(* CoDeSys 2.3.9.41 project: pns.pro *)
(* Libraries: STANDARD.LIB 4.10.05 10:14:46, IECSFC.LIB 13.4.06 14:51:28, SYSLIBTIME.LIB 20.2.06 13:31:16, SYSTASKINFO.LIB 20.2.06 13:31:38, ANALYZATION.LIB 5.10.99 08:05:06, SYSLIBCALLBACK.LIB 20.2.06 13:31:08, PID_Regulators.lib 28.12.06 17:47:54 *)

(* PLC configuration (modules and I/O channels)
Discrete input 6 bit [ID100] node 0, in %IB0 out %QB0 {Filtrationtime = 10; Filtrationtime = 10; Filtrationtime = 10; Filtrationtime = 10; Filtrationtime = 10; Filtrationtime = 10; Visibility = No; PinCount = 6; WatchDogPeriod = 1000; PollPeriod = 1}
  DI_ekmLower AT %IX0.0 [BitInput]
  DI_ekmUpper AT %IX0.1 [BitInput]
  DI_pmp1_auto AT %IX0.2 [BitInput]
  DI_pmp2_auto AT %IX0.3 [BitInput]
  DI_pmp3_auto AT %IX0.4 [BitInput]
  DI_fcAlarm AT %IX0.5 [BitInput]
Discrete output 4 bit [ID101] node 1, in %IB1 out %QB1 {PinCount = 4; SafeValueBool = FALSE; SafeValueBool = FALSE; SafeValueBool = FALSE; SafeValueBool = FALSE; Visibility = No}
  DO_fc_on AT %QX1.0 [BitOutput]
  DO_fc_run AT %QX1.1 [BitOutput]
  DO_lamp_fcAlarm AT %QX1.2 [BitOutput]
  DO_lamp_dryHod AT %QX1.3 [BitOutput]
Special output [ID104] node 2, in %IB2 out %QB2 {Visibility = No; PinCount = 1}
  AT %QX2.0 [BitOutput] Special output
Unifed signal sensor [ID700] node 3, in %IB3 out %QB3 {Type_of_sensor700 = IT_0_20; measure_interval = 0.5; ainlow = 0; ainhigh = 20; first_cor_point = 0; first_delta = 0; second_cor_point = 0; second_delta = 0; third_cor_point = 0; third_delta = 0; Visibility = No}
  AI_pres AT %ID3.0 [FloatInput] Value
  cirTime AT %IW3.1 [WordInput] Circular time
  Analog Input [ID107] node 0, in %IB3.0 out %QB3.0
Unifed signal sensor [ID700] node 4, in %IB4 out %QB4 {Type_of_sensor700 = IT_0_20; measure_interval = 0.5; ainlow = 0; ainhigh = 20; first_cor_point = 0; first_delta = 0; second_cor_point = 0; second_delta = 0; third_cor_point = 0; third_delta = 0; Visibility = No}
  AT %ID4.0 [FloatInput] Value
  AT %IW4.1 [WordInput] Circular time
  Analog Input [ID107] node 0, in %IB4.0 out %QB4.0
Unifed signal sensor [ID700] node 5, in %IB5 out %QB5 {Type_of_sensor700 = IT_0_20; measure_interval = 0.5; ainlow = 0; ainhigh = 20; first_cor_point = 0; first_delta = 0; second_cor_point = 0; second_delta = 0; third_cor_point = 0; third_delta = 0; Visibility = No}
  AT %ID5.0 [FloatInput] Value
  AT %IW5.1 [WordInput] Circular time
  Analog Input [ID107] node 0, in %IB5.0 out %QB5.0
Unifed signal sensor [ID700] node 6, in %IB6 out %QB6 {Type_of_sensor700 = IT_0_20; measure_interval = 0.5; ainlow = 0; ainhigh = 20; first_cor_point = 0; first_delta = 0; second_cor_point = 0; second_delta = 0; third_cor_point = 0; third_delta = 0; Visibility = No}
  AT %ID6.0 [FloatInput] Value
  AT %IW6.1 [WordInput] Circular time
  Analog Input [ID107] node 0, in %IB6.0 out %QB6.0
Analog output [ID106] node 7, in %IB7 out %QB7 {DAC_Type = Voltage 0-10 B; Analog_offset_correction = 0; Analog_full_range_correction = 0; SafeValueFloat = 0; Visibility = No}
  AO_ref AT %QD7.0 [FloatOutput] Value
Analog output [ID106] node 8, in %IB8 out %QB8 {DAC_Type = Voltage 0-10 B; Analog_offset_correction = 0; Analog_full_range_correction = 0; SafeValueFloat = 0; Visibility = No}
  AT %QD8.0 [FloatOutput] Value
ModBus (Master) [MODBUS_MASTER_ID450] node 9, in %IB9 out %QB9 {Visibility = No}
  AT %QD9.0 [DWordOutput] Last address
  AT %QW9.1 [WordOutput] Last error
  RS-485-1 [COM1_USART] node 0, in %IB9.0 out %QB9.0 {CommunicationSpeed = 19200; Parity = NO PARITY CHECK; BitLength = 8 bits; StopLength = One stop bit; InterfaceType = RS485; FrameOriented = RTU; Timeout = 0; Visibility = No}
  Universal Modbus device [ID2000] node 1, in %IB9.1 out %QB9.1 {ModuleIP = 10:0:0:223; ServiceTimeout = 150; TCPport = 502; NetMode = Serial; ModuleSlaveAddress = 2; RequestType = By poll time; PeriodOfService = 500; Visibility = No; RepeatCounter = 0; ByteSequence = Trace_mode}
    AT %QB9.1.0 [ComChannel] Command (0xff - Start)
PLC100_DI AT %IW9.1.0.0 [WordInput]
PLC100_DO AT %QW9.1.1.0 [WordOutput]
TCP [TCP_ID221] node 0, in %IB10.0.0 out %QB10.0.0 {RemotePort = 502; Visibility = No}
ktp_INPUT AT %QW10.1.0 [WordOutput] setTime, kaReset
ktp_OUTPUT AT %QW10.2.0 [WordOutput] pmp1,pmp2,pmp3,EKM,alarm,auto1,auto2,auto3
ktp_pressure AT %QW10.3.0 [WordOutput]
ktp_presStartDelta AT %QW10.4.0 [WordOutput]
ktp_presStopDelta AT %QW10.5.0 [WordOutput]
ktp_daySetpoint AT %QW10.6.0 [WordOutput]
ktp_nightSetpoint AT %QW10.7.0 [WordOutput]
ktp_finishSetpoint AT %QW10.8.0 [WordOutput]
ktp_pres4ma AT %QW10.9.0 [WordOutput]
ktp_pres20ma AT %QW10.10.0 [WordOutput]
ktp_startReserveDelay AT %QW10.11.0 [WordOutput]
ktp_stopReserveDelay AT %QW10.12.0 [WordOutput]
ktp_barToStartDirect AT %QW10.13.0 [WordOutput]
ktp_mainPmp AT %QW10.14.0 [WordOutput]
ktp_prop AT %QW10.15.0 [WordOutput]
ktp_integ AT %QW10.16.0 [WordOutput]
ktp_diff AT %QW10.17.0 [WordOutput]
ktp_integMin AT %QW10.18.0 [WordOutput]
ktp_integMax AT %QW10.19.0 [WordOutput]
ktp_dryHodDelay AT %QW10.20.0 [WordOutput]
ktp_aType_1 AT %QW10.21.0 [WordOutput]
ktp_aType_2 AT %QW10.22.0 [WordOutput]
ktp_aType_3 AT %QW10.23.0 [WordOutput]
ktp_aTime_1 AT %QW10.24.0 [WordOutput]
ktp_aTime_2 AT %QW10.25.0 [WordOutput]
ktp_aTime_3 AT %QW10.26.0 [WordOutput]
ktp_aDate_1 AT %QW10.27.0 [WordOutput]
ktp_aDate_2 AT %QW10.28.0 [WordOutput]
ktp_aDate_3 AT %QW10.29.0 [WordOutput]
ktp_aPres_1 AT %QW10.30.0 [WordOutput]
ktp_aPres_2 AT %QW10.31.0 [WordOutput]
ktp_aPres_3 AT %QW10.32.0 [WordOutput]
ktp_aSetpoint_1 AT %QW10.33.0 [WordOutput]
ktp_aSetpoint_2 AT %QW10.34.0 [WordOutput]
ktp_aSetpoint_3 AT %QW10.35.0 [WordOutput]
ktp_aFreq_1 AT %QW10.36.0 [WordOutput]
ktp_aFreq_2 AT %QW10.37.0 [WordOutput]
ktp_aFreq_3 AT %QW10.38.0 [WordOutput]
ktp_aCurr_1 AT %QW10.39.0 [WordOutput]
ktp_aCurr_2 AT %QW10.40.0 [WordOutput]
ktp_aCurr_3 AT %QW10.41.0 [WordOutput]
ktp_aMainPmp_1 AT %QW10.42.0 [WordOutput]
ktp_aMainPmp_2 AT %QW10.43.0 [WordOutput]
ktp_aMainPmp_3 AT %QW10.44.0 [WordOutput]
ktp_topPos AT %QW10.45.0 [WordOutput]
ktp_midPos AT %QW10.46.0 [WordOutput]
ktp_bottomPos AT %QW10.47.0 [WordOutput]
ktp_cursor AT %QW10.48.0 [WordOutput]
ktp_setHH AT %QW10.49.0 [WordOutput]
ktp_setMMin AT %QW10.50.0 [WordOutput]
ktp_setDD AT %QW10.51.0 [WordOutput]
ktp_setMM AT %QW10.52.0 [WordOutput]
ktp_setYYYY AT %QW10.53.0 [WordOutput]
ktp_currHH AT %QW10.54.0 [WordOutput]
ktp_currMMin AT %QW10.55.0 [WordOutput]
ktp_currDD AT %QW10.56.0 [WordOutput]
ktp_currMM AT %QW10.57.0 [WordOutput]
ktp_currYYYY AT %QW10.58.0 [WordOutput]
ktp_spHHday AT %QW10.59.0 [WordOutput]
ktp_spMMday AT %QW10.60.0 [WordOutput]
ktp_spHHnight AT %QW10.61.0 [WordOutput]
ktp_spMMnight AT %QW10.62.0 [WordOutput]
ktp_currFreq AT %QW10.63.0 [WordOutput]
ktp_currCurr AT %QW10.64.0 [WordOutput]
ktp_currPower AT %QW10.65.0 [WordOutput]
ktp_pmp1mode AT %QW10.66.0 [WordOutput]
ktp_pmp2mode AT %QW10.67.0 [WordOutput]
ktp_pmp3mode AT %QW10.68.0 [WordOutput]
AT %IW11.0 [WordInput] Cycle time in 100 mks
AT %IW11.1 [WordInput] Time to backup power down, s
AT %ID11.2 [FloatInput] Temp inside PLC
powerStatus AT %IX11.3 [BitInput] Power status
AT %IX11.4 [BitInput] CPU is overloaded, optimize your programm or increase PLC cycle
AT %IW11.5 [WordInput] Free processor resourse mks in 1 cycle
*)

(* Global variable list: Global_Variables *)
VAR_GLOBAL

	(* Times *)
	GetTime: CurTimeEx;
	TimeAndDate: SystemTimeDate;
	Sys_Time: SysTime64;

	(* Alarms *)
	Alarmy : WORD;

	sensBreak : BOOL; (* 1 *)
	sensShort : BOOL; (* 2 *)
	dryHod		 : BOOL; (* 3 *)
	ekmUpper : BOOL; (* 4 *)
	fcAlarm	: BOOL; (* 5 *)
	kaPmp1fc	: BOOL; (* 6 *)
	kaPmp2fc	: BOOL; (* 7 *)
	kaPmp3fc : BOOL; (* 8 *)
	kaKM1		: BOOL; (* 9 *)
END_VAR

(* POU PLC_PRG, ST *)
PROGRAM PLC_PRG
VAR
	NO_FIRST_PASS : BOOL := FALSE;

	(* Inputs *)
	pmp1_auto, pmp2_auto, pmp3_auto : BOOL;
	pmp1_state, pmp2_state, pmp3_state : BOOL;
	pmp1_stateD, pmp2_stateD, pmp3_stateD : BOOL;
	(*ekm_upper,*) ekm_lower : BOOL;

	(* Outputs *)
	pmp1fc, pmp2fc, pmp3fc : BOOL;
	pmp1d, pmp2d, pmp3d : BOOL;
	fc_on, fc_run : BOOL;

	(* Process *)
	dryTimer : TON;
	dryDelay : TIME;
	dryHodOk : BOOL;

	mainMustStart, secondMustStart, thirdMustStart : BOOL;

	pressure : WORD;
	daySetpoint, nightSetpoint, finishSetpoint : WORD; (* точность 0.01 *)
	presStartDelta, presStopDelta : WORD;
	startReserveDelay, stopReserveDelay : TIME;

	secondStartTimerGo, thirdStartTimerGo, secondStopTimerGo, thirdStopTimerGo : BOOL;
	secondStartTimer, thirdStartTimer, secondStopTimer, thirdStopTimer :TON;
	secondGo, thirdGo, secondStop, thirdStop : BOOL;
	mainStarted : BOOL;

	(* Reserve prepare *)
	secondPrepareToStart, secondPrepared : BOOL;
	barToStartDirect : WORD; (* точность 0.01 *)

	(* Priority *)
	mainPmp : WORD;
	pmp1_priority, pmp2_priority, pmp3_priority : WORD;

	(* Calibration *)
	pres4ma, pres20ma : WORD;

	(* SelectPump *)
	pmp1_mustRunFc, pmp2_mustRunFc, pmp3_mustRunFc : BOOL;
	(*pmp1_mustRunD, pmp2_mustRunD, pmp3_mustRunD : BOOL;*)
	secondStarted, thirdStarted : BOOL;

	(* PID *)
	lgPid : PID_FUNCTION;
	real_pres, real_setpoint, pid_out : REAL;
	prop, prop_r, diff : REAL;
	integ : DINT;
	integMin, integMax : REAL;

	(* Inverter *)
	inverterMustStart, inverterRun : BOOL;
	timerBeforeFcOn, timerBeforeFcRun : TON;
	fcCanOnByTimer, fcCanStartByTimer : BOOL;
	fcStartedWithPump1, fcStartedWithPump2, fcStartedWithPump3 : BOOL;

	inverterMustStop : BOOL;
	timerAfterFcStop, timerAfterFcOff : TON;
	fcByTimerStopped, fcByTimerSwitchedOff : BOOL;
	inverterSwitchedOff : BOOL;

	(* DryBlink *)
	dryHodDelay : TIME;
	offTimer, onTimer : TON;
	onLamp : BOOL;
	goBlink, goLight : BOOL;

	(* Alarmes *)
	breakDetect : BOOL;
	breakTimer : TON;

	shortDetect : BOOL;
	shortTimer : TON;

	fcAlarmDetect, fcAlarmFP : BOOL;
	fcAlarmTimer : TON;

	pmp1kaDetect, pmp2kaDetect, pmp3kaDetect : BOOL;
	pmp1kaTimer, pmp2kaTimer, pmp3kaTimer : TON;
	pmp1kaFP, pmp2kaFP, pmp3kaFP,  kmKaFP : BOOL;
	fc_state, fc_kaDetect : BOOL;
	fcKaTimer : TON;

	(* KA SPECIAL *)
	pmp1kaSave, pmp2kaSave, pmp3kaSave : BOOL;
	kaReset : BOOL;

	(* Times *)
	setTime : BOOL;
	pmp1_status: BOOL;

END_VAR
VAR RETAIN
	(* Process *)
	save_daySetpoint, save_nightSetpoint : WORD;
	save_spHHday, save_spMMday, save_spHHnight, save_spMMnight : WORD;
(*
	save_presStartDelta, save_presStopDelta : WORD;
	save_startReserveDelay, save_stopReserveDelay : WORD;
*)
(*
	(* Reserve prepare *)
	save_barToStartDirect : WORD;
*)
	(* Priority *)
	save_mainPmp : WORD;

	(* Calibration *)
	save_pres4ma, save_pres20ma : WORD;

	(* PID *)
	save_prop, save_diff : WORD;
	save_integ : WORD;
	save_integMin, save_integMax : WORD;
	save_analogOutMax : WORD;

	(* DryHod *)
	save_dryHodDelay : WORD;
	save : WORD;
	lg_freq, lg_curr, lg_pow : WORD;
END_VAR
(* доработать работу от ПЧ *)

IF NO_FIRST_PASS = FALSE THEN
			WithdrawRetain;
			inverterSwitchedOff := TRUE;
			NO_FIRST_PASS := TRUE;
END_IF;

Defaults;

SaveNewVal;

Times;

Inputs;

Calibration;

Setpoint;

Process;

DryLamp;
(*
SecondPrepare;
*)
Priority;

SelectPump;

PID;

InverterStarting;

InverterStopping;

Protect;

Alarmes;

Outputs;

ALARMS;

(* Block direct *)
pmp1d := FALSE;
pmp2d := FALSE;
pmp3d := FALSE;
END_PROGRAM
ACTION Alarmes:
(* SENS BREAK *)
IF AI_pres < 3.9 THEN
	breakDetect := TRUE;
ELSE
	breakDetect := FALSE;
END_IF;

breakTimer(IN:= breakDetect, PT:=T#1s, Q=>sensBreak, ET=> );


(* SENS SHORT *)
IF AI_pres > 21.0 THEN
	shortDetect := TRUE;
ELSE
	shortDetect := FALSE;
END_IF;

shortTimer(IN:= shortDetect, PT:=T#1s, Q=>sensShort, ET=> );

(* DRY HOD *) (* таймер в Process *)
dryHod := dryHodOk;

(* EKM UPPER *)

(* FC ALARM *)
IF DI_fcAlarm AND fc_on = TRUE THEN
	fcAlarmDetect := TRUE;
ELSE
	fcAlarmDetect := FALSE;
END_IF;

fcAlarmTimer(IN:= fcAlarmDetect, PT:=T#10s, Q=>fcAlarm, ET=> );

IF fcAlarm AND fcAlarmFP = FALSE THEN
	fcAlarmFP := TRUE;
	ShiftKtpMainPmp;
END_IF;

IF fcAlarm = FALSE THEN
	fcAlarmFP := FALSE;
END_IF;

(* PMP1 KA *)
IF pmp1fc AND pmp1_state = FALSE THEN
	pmp1kaDetect := TRUE;
ELSE
	pmp1kaDetect := FALSE;
END_IF;

pmp1kaTimer(IN:= pmp1kaDetect, PT:=T#10s, Q=>kaPmp1fc, ET=> );

IF kaPmp1fc AND pmp1kaFP = FALSE THEN
	pmp1kaFP := TRUE;
	pmp1kaSave := TRUE;
	ShiftKtpMainPmp;
END_IF;

IF kaPmp1fc = FALSE THEN
	pmp1kaFP := FALSE;
END_IF;

(* PMP2 KA *)
IF pmp2fc AND pmp2_state = FALSE THEN
	pmp2kaDetect := TRUE;
ELSE
	pmp2kaDetect := FALSE;
END_IF;

pmp2kaTimer(IN:= pmp2kaDetect, PT:=T#10s, Q=>kaPmp2fc, ET=> );

IF kaPmp2fc AND pmp2kaFP = FALSE THEN
	pmp2kaFP := TRUE;
	pmp2kaSave := TRUE;
	ShiftKtpMainPmp;
END_IF;

IF kaPmp2fc = FALSE THEN
	pmp2kaFP := FALSE;
END_IF;

(* PMP3 KA *)
IF pmp3fc AND pmp3_state = FALSE THEN
	pmp3kaDetect := TRUE;
ELSE
	pmp3kaDetect := FALSE;
END_IF;

pmp3kaTimer(IN:= pmp3kaDetect, PT:=T#10s, Q=>kaPmp3fc, ET=> );

IF kaPmp3fc AND pmp3kaFP = FALSE THEN
	pmp3kaFP := TRUE;
	pmp3kaSave := TRUE;
	ShiftKtpMainPmp;
END_IF;

IF kaPmp3fc = FALSE THEN
	pmp3kaFP := FALSE;
END_IF;

IF ktp_INPUT.1 THEN
	pmp1kaSave := FALSE;
	pmp2kaSave := FALSE;
	pmp3kaSave := FALSE;
	ktp_INPUT.1 := FALSE;
END_IF;

(* FC KA *)
IF fc_on AND fc_state = FALSE THEN
	fc_kaDetect := TRUE;
ELSE
	fc_kaDetect := FALSE;
END_IF;

fcKaTimer(IN:= fc_kaDetect, PT:=T#10s, Q=>kaKM1, ET=> );

IF kaKM1 AND kmKaFP = FALSE THEN
	kmKaFP := TRUE;
	ShiftKtpMainPmp;
END_IF;

IF kaKM1 = FALSE THEN
	kmKaFP := FALSE;
END_IF;

(* ALARMY *)
Alarmy.0 := sensBreak;
Alarmy.1 := sensShort;
Alarmy.2 := dryHod;

Alarmy.4 := fcAlarm;
Alarmy.5 := kaPmp1fc;
Alarmy.6 := kaPmp2fc;
Alarmy.7 := kaPmp3fc;
Alarmy.8 := kaKM1;

IF Alarmy > 0 THEN
	DO_lamp_fcAlarm := TRUE;
ELSE
	DO_lamp_fcAlarm := FALSE;
END_IF;
END_ACTION
ACTION Calibration:
pressure := pres4ma  + ( REAL_TO_WORD( AI_pres * 100 ) - 400 ) * ( pres20ma - pres4ma ) / 1600; (* wordpres := .... точность 0.01 *)

IF AI_pres < 4.0 THEN
	pressure := 0;
END_IF;
END_ACTION
ACTION Defaults:
IF ktp_daySetpoint = 0 THEN
	ktp_daySetpoint := 500;
END_IF;

IF ktp_nightSetpoint = 0 THEN
	ktp_nightSetpoint := 500;
END_IF;

IF ktp_pres20ma = 0 THEN
	ktp_pres20ma := 1000;
END_IF;

IF ktp_mainPmp = 0 THEN
	ktp_mainPmp := 2;
END_IF;

IF ktp_prop = 0 THEN
	ktp_prop := 30000;
END_IF;

IF ktp_integ = 0 THEN
	ktp_integ := 10;
END_IF;

IF ktp_spHHday = 0 THEN
	ktp_spHHday := 6;
END_IF;
END_ACTION
ACTION DryLamp:
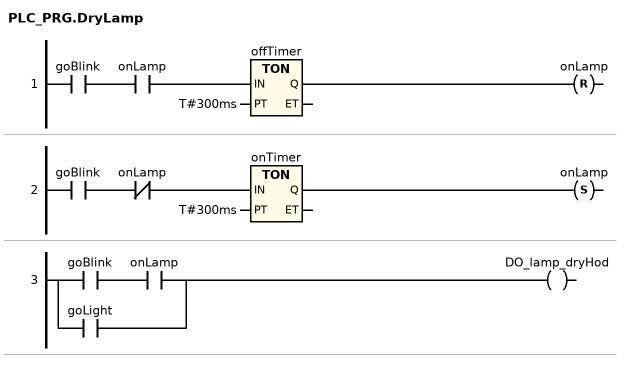
_LD_ (* Ladder Diagram *)
NETWORK 1
	[goBlink] - [onLamp] - offTimer:TON(IN: *, PT: T#300ms) --- (R onLamp)
NETWORK 2
	[goBlink] - [/onLamp] - onTimer:TON(IN: *, PT: T#300ms) --- (S onLamp)
NETWORK 3
	{ [goBlink] - [onLamp] | [goLight] } --- (DO_lamp_dryHod)
_END_LD_
(* the same logic as Structured Text *)
(* Network 1 *)
offTimer(IN := goBlink AND onLamp, PT := T#300ms);
IF offTimer.Q THEN onLamp := FALSE; END_IF;
(* Network 2 *)
onTimer(IN := goBlink AND NOT onLamp, PT := T#300ms);
IF onTimer.Q THEN onLamp := TRUE; END_IF;
(* Network 3 *)
DO_lamp_dryHod := goBlink AND onLamp OR goLight;
END_ACTION
ACTION Inputs:
(* OWEN100 *)
pmp1_auto := DI_pmp1_auto;
pmp2_auto := DI_pmp2_auto;
pmp3_auto := DI_pmp3_auto;

pmp1_state := PLC100_DI.0;
pmp2_state := PLC100_DI.1;
pmp3_state := PLC100_DI.2;

fc_state := PLC100_DI.3;

pmp1_stateD := PLC100_DI.4;
pmp2_stateD := PLC100_DI.5;
pmp3_stateD := PLC100_DI.6;

(* OWEN150 *)
ekm_lower := DI_ekmLower;

(* Process *)
daySetpoint := ktp_daySetpoint;
nightSetpoint := ktp_nightSetpoint;
startReserveDelay := WORD_TO_TIME ( 1000 * ktp_startReserveDelay );
stopReserveDelay := WORD_TO_TIME ( 1000 * ktp_stopReserveDelay );
presStartDelta := ktp_presStartDelta;
presStopDelta := ktp_presStopDelta;

(* Reserve prepare *)
barToStartDirect := ktp_barToStartDirect;

(* Priority *)
IF mainPmp <> ktp_mainPmp THEN
	secondMustStart := FALSE;
	thirdMustStart := FALSE;
	IF secondStarted = FALSE AND thirdStarted = FALSE THEN
		mainPmp := ktp_mainPmp;
	END_IF;
END_IF;

(* Calibration *)
pres4ma := ktp_pres4ma;
pres20ma := ktp_pres20ma;

(* PID *)
prop := WORD_TO_REAL( ktp_prop ) / 100;
integ := ktp_integ;
diff := WORD_TO_REAL( ktp_diff ) / 100;
integMin := WORD_TO_REAL( ktp_integMin ) / 100;
integMax := WORD_TO_REAL( ktp_integMax ) / 100;

(* Dry hod *)
dryHodDelay := WORD_TO_TIME ( 1000 * ktp_dryHodDelay );
END_ACTION
ACTION InverterStarting:
IF inverterSwitchedOff AND mainMustStart THEN
	inverterMustStart := TRUE;
	IF pmp1_mustRunFc THEN
		pmp1fc := TRUE;
	ELSE
		IF pmp2_mustRunFc THEN
			pmp2fc := TRUE;
		ELSE
			IF pmp3_mustRunFc THEN
				pmp3fc := TRUE;
			END_IF;
		END_IF
	END_IF;
END_IF;

IF pmp1_mustRunFc = FALSE AND pmp2_mustRunFc = FALSE AND pmp3_mustRunFc = FALSE THEN
	inverterMustStart := FALSE;
END_IF;

timerBeforeFcOn(IN:=inverterMustStart, PT:=T#10s, Q=>fcCanOnByTimer, ET=> );

IF fcCanOnByTimer THEN
	fc_on := TRUE;
END_IF;

timerBeforeFcRun(IN:=fcCanOnByTimer, PT:=T#10s, Q=>fcCanStartByTimer, ET=> );

IF fcCanStartByTimer THEN
	inverterMustStart := FALSE;
	inverterSwitchedOff := FALSE;
	mainStarted := TRUE;
	IF pmp1fc AND pmp2fc = FALSE AND pmp3fc = FALSE THEN
		fc_run := TRUE;
		inverterRun := TRUE;
		fcStartedWithPump1 := TRUE;
	ELSE
		IF pmp2fc AND pmp1fc = FALSE AND pmp3fc = FALSE THEN
			fc_run := TRUE;
			inverterRun := TRUE;
			fcStartedWithPump2 := TRUE;
		ELSE
			IF pmp3fc AND pmp1fc = FALSE AND pmp2fc = FALSE THEN
				fc_run := TRUE;
				inverterRun := TRUE;
				fcStartedWithPump3 := TRUE;
			ELSE
				inverterMustStop := TRUE;
			END_IF;
		END_IF;
	END_IF;
END_IF;
END_ACTION
ACTION InverterStopping:
IF inverterRun THEN
	IF mainMustStart = FALSE THEN
		inverterMustStop := TRUE;
	END_IF;

	IF pmp1_auto = FALSE AND pmp2_auto = FALSE AND pmp3_auto = FALSE THEN
		inverterMustStop := TRUE;
	END_IF;

	IF pmp1_mustRunFc AND (fcStartedWithPump2 OR fcStartedWithPump3) THEN
		inverterMustStop := TRUE;
	END_IF;

	IF pmp2_mustRunFc AND (fcStartedWithPump1 OR fcStartedWithPump3) THEN
		inverterMustStop := TRUE;
	END_IF;

	IF pmp3_mustRunFc AND (fcStartedWithPump2 OR fcStartedWithPump1) THEN
		inverterMustStop := TRUE;
	END_IF;

	IF inverterMustStop THEN
		fc_run := FALSE;
	END_IF;
END_IF;

timerAfterFcStop(IN:= inverterMustStop, PT:=T#14s, Q=>fcByTimerStopped, ET=> );

IF fcByTimerStopped THEN
	fc_on := FALSE;
END_IF;

timerAfterFcOff(IN:= fcByTimerStopped, PT:=T#40s, Q=>fcByTimerSwitchedOff, ET=> );

IF fcByTimerSwitchedOff THEN
	inverterSwitchedOff := TRUE;

	inverterMustStop := FALSE;
	mainStarted := FALSE;
	pmp1fc := FALSE;
	pmp2fc := FALSE;
	pmp3fc := FALSE;
	pmp1_mustRunFc := FALSE;
	pmp2_mustRunFc := FALSE;
	pmp3_mustRunFc := FALSE;
	fcStartedWithPump1 := FALSE;
	fcStartedWithPump2 := FALSE;
	fcStartedWithPump3 := FALSE;
	inverterRun := FALSE;
END_IF;
END_ACTION
ACTION Outputs:
PLC100_DO.0 := pmp1fc;
PLC100_DO.1 := pmp2fc;
PLC100_DO.2 := pmp3fc;

PLC100_DO.3 := pmp1d;
PLC100_DO.4 := pmp2d;
PLC100_DO.5 := pmp3d;

DO_fc_on := fc_on;
DO_fc_run := fc_run;

ktp_finishSetpoint := finishSetpoint;
ktp_pressure := pressure;


ktp_currHH := TimeAndDate.Hour;
ktp_currMMin := TimeAndDate.Minute;

ktp_currDD := TimeAndDate.Day;
ktp_currMM := TimeAndDate.Month;
ktp_currYYYY := TimeAndDate.Year;

ktp_OUTPUT.0 := pmp1_state;
ktp_OUTPUT.1 := pmp2_state;
ktp_OUTPUT.2 := pmp3_state;
ktp_OUTPUT.3 := DI_ekmLower;
IF Alarmy > 0 THEN
	ktp_OUTPUT.4 := TRUE;
ELSE
	ktp_OUTPUT.4 := FALSE;
END_IF;
ktp_OUTPUT.5 := pmp1_auto;
ktp_OUTPUT.6 := pmp2_auto;
ktp_OUTPUT.7 := pmp3_auto;

ktp_currFreq := lg_freq;
ktp_currCurr := lg_curr;
ktp_currPower := lg_pow;

ktp_OUTPUT.8 := pmp1kaSave;
ktp_OUTPUT.9 := pmp2kaSave;
ktp_OUTPUT.10 := pmp3kaSave;

(* pmp modes *)
IF pmp1_state = FALSE AND pmp1_stateD = FALSE THEN
	ktp_pmp1mode := 1;
ELSE
	IF pmp1_state THEN
		ktp_pmp1mode := 2;
	END_IF;
	IF pmp1_stateD THEN
		ktp_pmp1mode := 3;
	END_IF;
END_IF;

IF pmp2_state = FALSE AND pmp2_stateD = FALSE THEN
	ktp_pmp2mode := 1;
ELSE
	IF pmp2_state THEN
		ktp_pmp2mode := 2;
	END_IF;
	IF pmp2_stateD THEN
		ktp_pmp2mode := 3;
	END_IF;
END_IF;

IF pmp3_state = FALSE AND pmp3_stateD = FALSE THEN
	ktp_pmp3mode := 1;
ELSE
	IF pmp3_state THEN
		ktp_pmp3mode := 2;
	END_IF;
	IF pmp3_stateD THEN
		ktp_pmp3mode := 3;
	END_IF;
END_IF;
END_ACTION
ACTION PID:
IF sensBreak = FALSE AND sensShort = FALSE THEN

	real_pres := WORD_TO_REAL( pressure ) / 100;
	real_setpoint := WORD_TO_REAL( finishSetpoint ) / 100;

	prop_r := prop / 100;

	lgPid(
		PV:= real_pres , (* REAL Входное значение*)
		PV_TIME:= cirTime, (* WORD Время получения входной величины - отсчитвыается в долях секунды и берется из UNIVERSAL Sensor/ Circular time*)
		SP:= real_setpoint , (* REAL уставка*)
		PB:= prop_r, (*REAL полоса пропорциональности*)
		TI_:= integ, (* DINT постоянная интегрирования - 4 байтовое целое знаковое*)
		TD_:= diff, (* REAL постоянная диффереренцирования*)
		_IMIN:= -1.0, (* REAL минимум интегральной составляющей*)
		_IMAX:= 1.0, (* REAL максимум интегральной составляющей*)
		OUT_VAL=> pid_out); (* REAL Выходное значение*)

	(*analogOutMax := WORD_TO_REAL( ktp_analogOutMax ) / 100;*)

	(*IF analogOutMax <= 10.0 THEN*)
		AO_ref := ( pid_out + 100 ) * 0.05;
	(*END_IF;*)
ELSE
	AO_ref := 6.0;
END_IF;
END_ACTION
ACTION Priority:
IF pmp1_auto OR pmp2_auto OR pmp3_auto THEN

IF mainPmp = 1 THEN
	IF pmp1_auto = FALSE THEN
		ShiftKtpMainPmp;
	ELSE
		pmp1_priority := 1;
		IF pmp3_auto = TRUE THEN
			pmp3_priority := 2;
			IF pmp2_auto = TRUE THEN
				pmp2_priority := 3;
			ELSE
				pmp2_priority := 4;
			END_IF;
		ELSE
			pmp3_priority := 4;
			IF pmp2_auto = TRUE THEN
				pmp2_priority := 2;
			ELSE
				pmp2_priority := 4;
			END_IF;
		END_IF;
	END_IF;
END_IF;


IF mainPmp = 2 THEN
	IF pmp2_auto = FALSE THEN
		ShiftKtpMainPmp;
	ELSE
		pmp2_priority := 1;
		IF pmp1_auto = TRUE THEN
			pmp1_priority := 2;
			IF pmp3_auto = TRUE THEN
				pmp3_priority := 3;
			ELSE
				pmp3_priority := 4;
			END_IF;
		ELSE
			pmp1_priority := 4;
			IF pmp3_auto = TRUE THEN
				pmp3_priority := 2;
			ELSE
				pmp3_priority := 4;
			END_IF;
		END_IF;
	END_IF;
END_IF;


IF mainPmp = 3 THEN
	IF pmp3_auto = FALSE THEN
		ShiftKtpMainPmp;
	ELSE
		pmp3_priority := 1;
		IF pmp2_auto = TRUE THEN
			pmp2_priority := 2;
			IF pmp1_auto = TRUE THEN
				pmp1_priority := 3;
			ELSE
				pmp1_priority := 4;
			END_IF;
		ELSE
			pmp2_priority := 4;
			IF pmp1_auto = TRUE THEN
				pmp1_priority := 2;
			ELSE
				pmp1_priority := 4;
			END_IF;
		END_IF;
	END_IF;
END_IF;

END_IF;
END_ACTION
ACTION Process:
IF ekm_lower THEN
	goBlink := TRUE;
ELSE
	goBlink := FALSE;
	goLight := FALSE;
END_IF;

dryTimer(IN:= ekm_lower, PT:=dryHodDelay, Q=>dryHodOk, ET=> );

(* условия включения основного НА *)
IF dryHodOk = FALSE THEN
	mainMustStart := TRUE;
ELSE
	goLight := TRUE;
	mainMustStart := FALSE;
	secondMustStart := FALSE;
	thirdMustStart := FALSE;
END_IF;

(*
(* включение резервного НА *)
(* IF ( UINT_TO_REAL ( mainFreq ) / 100 >  freqLimStart  )  AND *)
IF ( presStartDelta < finishSetpoint - pressure ) AND mainStarted
	THEN secondStartTimerGo := TRUE;
	ELSE secondStartTimerGo := FALSE;
END_IF;


secondStartTimer(IN:= secondStartTimerGo, PT:=startReserveDelay, Q=>secondGo, ET=> );

IF secondGo THEN
	secondPrepareToStart := TRUE;
END_IF;

IF secondPrepareToStart THEN
	secondPrepare;
END_IF;

IF secondPrepared THEN
	secondMustStart := TRUE;
	secondPrepared := FALSE;
	secondPrepareToStart := FALSE;
END_IF;

(* выключение резервного НА *)
IF ( presStopDelta < pressure - finishSetpoint )
	THEN secondStopTimerGo := TRUE;
	ELSE secondStopTimerGo := FALSE;
END_IF;

secondStopTimer(IN:= secondStopTimerGo, PT:=stopReserveDelay, Q=>secondStop, ET=> );

IF secondStop OR mainMustStart = FALSE THEN
	secondMustStart := FALSE;
END_IF;
*)
END_ACTION
ACTION Protect:
IF pmp1fc THEN
	pmp1d := FALSE;
	pmp2fc := FALSE;
	pmp3fc := FALSE;
END_IF;

IF pmp2fc THEN
	pmp2d := FALSE;
	pmp1fc := FALSE;
	pmp3fc := FALSE;
END_IF;

IF pmp3fc THEN
	pmp3d := FALSE;
	pmp2fc := FALSE;
	pmp1fc := FALSE;
END_IF;
END_ACTION
ACTION SaveNewVal:
(* Process *)
IF save_daySetpoint <> ktp_daySetpoint
	THEN save_daySetpoint := ktp_daySetpoint;
END_IF;

IF save_nightSetpoint <> ktp_nightSetpoint
	THEN save_nightSetpoint := ktp_nightSetpoint;
END_IF;

IF save_spHHday <> ktp_spHHday
	THEN save_spHHday := ktp_spHHday;
END_IF;

IF save_spMMday <> ktp_spMMday
	THEN save_spMMday := ktp_spMMday;
END_IF;

IF save_spHHnight <> ktp_spHHnight
	THEN save_spHHnight := ktp_spHHnight;
END_IF;

IF save_spMMnight <> ktp_spMMnight
	THEN save_spMMnight := ktp_spMMnight;
END_IF;
(*
IF save_startReserveDelay <> ktp_startReserveDelay
	THEN save_startReserveDelay := ktp_startReserveDelay;
END_IF;

IF save_stopReserveDelay <> ktp_stopReserveDelay
	THEN save_stopReserveDelay := ktp_stopReserveDelay;
END_IF;

IF save_presStartDelta <> ktp_presStartDelta
	THEN save_presStartDelta := ktp_presStartDelta;
END_IF;

IF save_presStopDelta <> ktp_presStopDelta
	THEN save_presStopDelta := ktp_presStopDelta;
END_IF;
*)
(* Reserve prepare *)
(*
IF save_barToStartDirect <> ktp_barToStartDirect
	THEN save_barToStartDirect := ktp_barToStartDirect;
END_IF;
*)
(* Priority *)
IF save_mainPmp <> ktp_mainPmp
	THEN save_mainPmp := ktp_mainPmp;
END_IF;

(* Calibration *)
IF save_pres4ma <> ktp_pres4ma
	THEN save_pres4ma := ktp_pres4ma;
END_IF;

IF save_pres20ma <> ktp_pres20ma
	THEN save_pres20ma := ktp_pres20ma;
END_IF;

(* PID *)
IF save_prop <> ktp_prop
	THEN save_prop := ktp_prop;
END_IF;

IF save_diff <> ktp_diff
	THEN save_diff := ktp_diff;
END_IF;

IF save_integ <> ktp_integ
	THEN save_integ := ktp_integ;
END_IF;

IF save_integMin <> ktp_integMin
	THEN save_integMin := ktp_integMin;
END_IF;

IF save_integMax <> ktp_integMax
	THEN save_integMax := ktp_integMax;
END_IF;

(* Dry Hod *)
IF save_dryHodDelay <> ktp_dryHodDelay
	THEN save_dryHodDelay := ktp_dryHodDelay;
END_IF;
END_ACTION
ACTION SecondPrepare:
finishSetpoint := 0;

IF ( pressure < barToStartDirect ) THEN
	secondPrepared := TRUE;
END_IF;
END_ACTION
ACTION SelectPump:
(* НА 1 *)

IF pmp1_auto THEN
	IF pmp1_priority = 1  THEN
		IF mainMustStart THEN
			pmp1_mustRunFc := TRUE;
		ELSE
			pmp1_mustRunFc := FALSE;
		END_IF;
	END_IF;

	IF pmp1_priority = 2 THEN
		IF secondMustStart THEN
			pmp1d := TRUE;
			secondStarted := TRUE;
		ELSE
			pmp1d := FALSE;
			secondStarted := FALSE;
		END_IF;
	END_IF;

	IF pmp1_priority = 3 THEN
		IF thirdMustStart THEN
			pmp1d := TRUE;
			thirdStarted := TRUE;
		ELSE
			pmp1d := FALSE;
			thirdStarted := FALSE;
		END_IF;
	END_IF;
ELSE
	pmp1_mustRunFc := FALSE;
	pmp1d := FALSE;
	IF pmp1_priority = 2 THEN
		secondStarted := FALSE;
	END_IF;
	IF pmp1_priority = 3 THEN
		thirdStarted := FALSE;
	END_IF;
END_IF;

IF pmp1_auto = FALSE THEN
	pmp1d := FALSE;
END_IF;

(* НА 2 *)

IF pmp2_auto THEN
	IF pmp2_priority = 1 THEN
		IF mainMustStart THEN
			pmp2_mustRunFc := TRUE;
		ELSE
			pmp2_mustRunFc := FALSE;
		END_IF;
	END_IF;

	IF pmp2_priority = 2 THEN
		IF secondMustStart THEN
			pmp2d := TRUE;
			secondStarted := TRUE;
		ELSE
			pmp2d := FALSE;
			secondStarted := FALSE;
		END_IF;
	END_IF;

	IF pmp2_priority = 3 THEN
		IF thirdMustStart THEN
			pmp2d := TRUE;
			thirdStarted := TRUE;
		ELSE
			pmp2d := FALSE;
			thirdStarted := FALSE;
		END_IF;
	END_IF;
ELSE
	pmp2_mustRunFc := FALSE;
	pmp2d := FALSE;
	IF pmp2_priority = 2 THEN
		secondStarted := FALSE;
	END_IF;
	IF pmp2_priority = 3 THEN
		thirdStarted := FALSE;
	END_IF;
END_IF;

IF pmp2_auto = FALSE THEN
	pmp2d := FALSE;
END_IF;

(* НА 3 *)

IF pmp3_auto THEN
	IF pmp3_priority = 1 THEN
		IF mainMustStart THEN
			pmp3_mustRunFc := TRUE;
		ELSE
			pmp3_mustRunFc := FALSE;
		END_IF;
	END_IF;

	IF pmp3_priority = 2 THEN
		IF secondMustStart THEN
			pmp3d := TRUE;
			secondStarted := TRUE;
		ELSE
			pmp3d := FALSE;
			secondStarted := FALSE;
		END_IF;
	END_IF;

	IF pmp3_priority = 3 THEN
		IF thirdMustStart THEN
			pmp3d := TRUE;
			thirdStarted := TRUE;
		ELSE
			pmp3d := FALSE;
			thirdStarted := FALSE;
		END_IF;
	END_IF;
ELSE
	pmp3_mustRunFc := FALSE;
	pmp3d := FALSE;
	IF pmp3_priority = 2 THEN
		secondStarted := FALSE;
	END_IF;
	IF pmp3_priority = 3 THEN
		thirdStarted := FALSE;
	END_IF;
END_IF;

IF pmp3_auto = FALSE THEN
	pmp3d := FALSE;
END_IF;
END_ACTION
ACTION Setpoint:
IF ktp_spHHnight > ktp_spHHday THEN
	IF TimeAndDate.Hour = ktp_spHHnight AND TimeAndDate.Minute >= ktp_spMMnight THEN
		finishSetpoint := nightSetpoint;
	END_IF;
	IF TimeAndDate.Hour >ktp_spHHnight AND TimeAndDate.Hour > ktp_spHHday THEN
		finishSetpoint := nightSetpoint;
	END_IF;
	IF TimeAndDate.Hour >= 0 AND TimeAndDate.Hour < ktp_spHHday THEN
		finishSetpoint := nightSetpoint;
	END_IF;
	IF TimeAndDate.Hour = ktp_spHHday AND TimeAndDate.Minute < ktp_spMMday THEN
		finishSetpoint := nightSetpoint;
	END_IF;
	IF TimeAndDate.Hour = ktp_spHHday AND TimeAndDate.Minute >= ktp_spMMday THEN
		finishSetpoint := daySetpoint;
	END_IF;
	IF TimeAndDate.Hour > ktp_spHHday AND TimeAndDate.Hour < ktp_spHHnight THEN
		finishSetpoint := daySetpoint;
	END_IF;
	IF TimeAndDate.Hour = ktp_spHHnight AND TimeAndDate.Minute < ktp_spMMnight THEN
		finishSetpoint := daySetpoint;
	END_IF;
END_IF;

IF ktp_spHHnight < ktp_spHHday THEN
	IF TimeAndDate.Hour = ktp_spHHnight AND TimeAndDate.Minute >= ktp_spMMnight THEN
		finishSetpoint := nightSetpoint;
	END_IF;
	IF TimeAndDate.Hour > ktp_spHHnight AND TimeAndDate.Hour < ktp_spHHday THEN
		finishSetpoint := nightSetpoint;
	END_IF;
	IF TimeAndDate.Hour = ktp_spHHday AND TimeAndDate.Minute < ktp_spMMday THEN
		finishSetpoint := nightSetpoint;
	END_IF;
	IF TimeAndDate.Hour = ktp_spHHday AND TimeAndDate.Minute >= ktp_spMMday THEN
		finishSetpoint := daySetpoint;
	END_IF;
	IF TimeAndDate.Hour > ktp_spHHday THEN
		finishSetpoint := daySetpoint;
	END_IF;
	IF TimeAndDate.Hour >= 0 AND ktp_spHHnight > 0 THEN
		finishSetpoint := daySetpoint;
	END_IF;
	IF TimeAndDate.Hour = ktp_spHHnight AND TimeAndDate.Minute < ktp_spMMnight THEN
		finishSetpoint := daySetpoint;
	END_IF;
END_IF;

(*
IF TimeAndDate.Hour = ktp_spHHnight AND TimeAndDate.Minute = ktp_spMMnight AND THEN
	finishSetpoint := nightSetpoint;
END_IF;

IF TimeAndDate.Hour = ktp_spHHday AND TimeAndDate.Minute = ktp_spMMday AND TimeAndDate.Second = 0 THEN
	finishSetpoint := daySetpoint;
END_IF;
*)
END_ACTION
ACTION ShiftKtpMainPmp:
ktp_mainPmp := ktp_mainPmp + 1;

IF ktp_mainPmp > 3 OR ktp_mainPmp = 0 THEN
	ktp_mainPmp := 1;
END_IF;
END_ACTION
ACTION Times:
TimeAndDate.Day :=0;
TimeAndDate.DayOfWeek :=0;
TimeAndDate.dwHighMsec :=0;
TimeAndDate.dwLowMSecs :=0;
TimeAndDate.Milliseconds :=0;
TimeAndDate.Minute :=0;
TimeAndDate.Second :=0;
TimeAndDate.Hour :=0;
TimeAndDate.Year :=0;
TimeAndDate.Month :=0;
Sys_time.ulHigh :=0;
Sys_time.ulLow :=0;
GetTime (SystemTime:=Sys_Time , TimeDate:= TimeAndDate);


IF ktp_INPUT.0 THEN
	TimeAndDate.Minute:=ktp_setMMin;
	TimeAndDate.Second:=10;
	TimeAndDate.Hour:=ktp_setHH;
	TimeAndDate.Day:=ktp_setDD;
	TimeAndDate.Month:=ktp_setMM;
	TimeAndDate.Year:=ktp_setYYYY;
	GetTime (SystemTime:=Sys_Time , TimeDate:= TimeAndDate);

	ktp_INPUT.0 := FALSE;
END_IF;
END_ACTION
ACTION WithdrawRetain:
(* Process *)
ktp_daySetpoint := save_daySetpoint;
ktp_nightSetpoint := save_nightSetpoint;
ktp_spHHday := save_spHHday;
ktp_spMMday := save_spMMday;
ktp_spHHnight := save_spHHnight;
ktp_spMMnight := save_spMMnight;
(*
ktp_startReserveDelay := save_startReserveDelay;
ktp_stopReserveDelay := save_stopReserveDelay;
ktp_presStartDelta := save_presStartDelta;
ktp_presStopDelta := save_presStopDelta;
*)
(*
(* Reserve prepare *)
ktp_barToStartDirect := save_barToStartDirect;
*)
(* Priority *)
ktp_mainPmp := save_mainPmp;

(* Calibration *)
ktp_pres4ma := save_pres4ma;
ktp_pres20ma := save_pres20ma;

(* PID *)
ktp_prop := save_prop;
ktp_diff := save_diff;
ktp_integ := save_integ;
ktp_integMin := save_integMin;
ktp_integMax := save_integMax;

(* Dry hod *)
ktp_dryHodDelay := save_dryHodDelay;
END_ACTION

(* POU ALARMS, ST *)
PROGRAM ALARMS
VAR
	fp_sensBreak : BOOL; (* 1 *)
	fp_sensShort  : BOOL; (* 2 *)
	fp_ekmLower  : BOOL; (* 3 *)
	fp_ekmUpper  : BOOL; (* 4 *)
	fp_fcAlarm		 : BOOL; (* 5 *)
	fp_kaPmp1fc	 : BOOL; (* 6 *)
	fp_kaPmp2fc	 : BOOL; (* 7 *)
	fp_kaPmp3fc 	 : BOOL; (* 8 *)
	fp_kaKM1		 : BOOL; (* 9 *)
	aPowerOffFP 	: BOOL; (* 10 *)

	last_aType 	:  WORD;

	topPos, midPos, bottomPos : INT;


END_VAR
VAR RETAIN
	id	: INT;
	(* must be retain *)
	aType 		: ARRAY[0..99] OF WORD;
	aTime 		: ARRAY[0..99] OF WORD;
	aDate 		: ARRAY[0..99] OF WORD;
	pres		: ARRAY[0..99] OF WORD;
	setpoint	: ARRAY[0..99] OF WORD;
	freq		: ARRAY[0..99] OF WORD;
	curr		: ARRAY[0..99] OF WORD;
	mainPmp 	: ARRAY[0..99] OF WORD;

END_VAR
last_aType := 0;

IF ktp_cursor = 127 THEN
	PutCursorToLastAlarm;
END_IF

CorrectCursor;

FillFields;

Check;

ktp_topPos := INT_TO_WORD( topPos );
ktp_midPos := INT_TO_WORD( midPos );
ktp_bottomPos := INT_TO_WORD( bottomPos );
END_PROGRAM
ACTION AddNew:
aType[ id ] := last_aType;
aTime[ id ] := TimeAndDate.Hour * 100 + TimeAndDate.Minute;
aDate[ id ] := TimeAndDate.Day * 100 + TimeAndDate.Month;
pres[ id ] := ktp_pressure;
setpoint[ id ] := ktp_finishSetpoint;
freq[ id ] := 0;
curr[ id ] := 0;
mainPmp[ id ] := ktp_mainPmp;

id := id + 1;

IF id >= 100 THEN
	id := 0;
END_IF;

ktp_cursor := INT_TO_WORD( id );
END_ACTION
ACTION Check:
(* SENS BREAK *)
IF sensBreak AND fp_sensBreak = FALSE THEN
	fp_sensBreak := TRUE;
	last_aType := 1;
	AddNew;
END_IF;

IF sensBreak = FALSE THEN
	fp_sensBreak := FALSE;
END_IF;

(* SENS SHORT *)
IF sensShort AND fp_sensShort = FALSE THEN
	fp_sensShort := TRUE;
	last_aType := 2;
	AddNew;
END_IF;

IF sensShort = FALSE THEN
	fp_sensShort := FALSE;
END_IF;

(* EKM LOWER *)
IF dryHod AND fp_ekmLower = FALSE THEN
	fp_ekmLower := TRUE;
	last_aType := 3;
	AddNew;
END_IF;

IF dryHod = FALSE THEN
	fp_ekmLower := FALSE;
END_IF;

(* EKM UPPER *)
IF ekmUpper AND fp_ekmUpper = FALSE THEN
	fp_ekmUpper := TRUE;
	last_aType := 4;
	AddNew;
END_IF;

IF ekmUpper = FALSE THEN
	fp_ekmUpper := FALSE;
END_IF;

(* FC ALARM *)
IF fcAlarm AND fp_fcAlarm = FALSE THEN
	fp_fcAlarm := TRUE;
	last_aType := 5;
	AddNew;
END_IF;

IF fcAlarm = FALSE THEN
	fp_fcAlarm := FALSE;
END_IF;

(* KA PMP1FC *)
IF kaPmp1fc AND fp_kaPmp1fc = FALSE THEN
	fp_kaPmp1fc := TRUE;
	last_aType := 6;
	AddNew;
END_IF;

IF kaPmp1fc = FALSE THEN
	fp_kaPmp1fc := FALSE;
END_IF;

(* KA PMP2FC *)
IF kaPmp2fc AND fp_kaPmp2fc = FALSE THEN
	fp_kaPmp2fc := TRUE;
	last_aType := 7;
	AddNew;
END_IF;

IF kaPmp2fc = FALSE THEN
	fp_kaPmp2fc := FALSE;
END_IF;

(* KA PMP3FC *)
IF kaPmp3fc AND fp_kaPmp3fc = FALSE THEN
	fp_kaPmp3fc := TRUE;
	last_aType := 8;
	AddNew;
END_IF;

IF kaPmp3fc = FALSE THEN
	fp_kaPmp3fc := FALSE;
END_IF;

(* KA KM1 *)
IF kaKM1 AND fp_kaKM1 = FALSE THEN
	fp_kaKM1 := TRUE;
	last_aType := 9;
	AddNew;
END_IF;

IF kaKM1 = FALSE THEN
	fp_kaKM1 := FALSE;
END_IF;

(* POWER *)
IF powerStatus = FALSE AND aPowerOffFP = FALSE  THEN
	aPowerOffFP := TRUE;
	last_aType := 10;
	AddNew;
END_IF;

IF powerStatus THEN
	aPowerOffFP := FALSE;
END_IF;
END_ACTION
ACTION CorrectCursor:
IF ktp_cursor > 99 THEN
	ktp_cursor := 0;
END_IF;

topPos := ktp_cursor;

midPos := ktp_cursor - 1;

bottomPos := ktp_cursor - 2;

IF ktp_cursor = 0 THEN
	midPos := 99;
	bottomPos := 98;
END_IF;

IF ktp_cursor = 1 THEN
	bottomPos := 99;
END_IF;
END_ACTION
ACTION FillFields:
ktp_aType_1 		:= aType		[ topPos ];
ktp_aTime_1 		:= aTime		[ topPos ];
ktp_aDate_1 		:= aDate		[ topPos ];
ktp_aPres_1 		:= pres			[ topPos ];
ktp_aSetpoint_1	 := setpoint	[ topPos ];
ktp_aFreq_1 		:= freq			[ topPos ];
ktp_aCurr_1	 	:= curr			[ topPos ];
ktp_aMainPmp_1 := mainPmp	[ topPos ];

ktp_aType_2 		:= aType		[ midPos ];
ktp_aTime_2 		:= aTime		[ midPos ];
ktp_aDate_2		:= aDate		[ midPos ];
ktp_aPres_2 		:= pres			[ midPos ];
ktp_aSetpoint_2 	:= setpoint		[ midPos ];
ktp_aFreq_2 		:= freq			[ midPos ];
ktp_aCurr_2 		:= curr			[ midPos ];
ktp_aMainPmp_2 := mainPmp	[ midPos ];

ktp_aType_3 		:= aType		[ bottomPos ];
ktp_aTime_3 		:= aTime		[ bottomPos ];
ktp_aDate_3		:= aDate		[ bottomPos ];
ktp_aPres_3 		:= pres			[ bottomPos ];
ktp_aSetpoint_3 	:= setpoint		[ bottomPos ];
ktp_aFreq_3 		:= freq			[ bottomPos ];
ktp_aCurr_3 		:= curr			[ bottomPos ];
ktp_aMainPmp_3 := mainPmp	[ bottomPos ];
END_ACTION
ACTION PutCursorToLastAlarm:
ktp_cursor := INT_TO_WORD( id ) - 1;
END_ACTION
